INTERFACE Queryable EXTENDS __SYSTEM.IQueryInterface

END_INTERFACE

(* stored: Version 1.1.0.1
   Itf Queryable: Id {b9eb6f36-0420-4aac-a46a-035e38d7498b} *)
